(* CoDeSys 2.3 export: TUZSIGNAL.EXP *)

(* Data type *)
TYPE tUZSignal : REAL;
END_TYPE
